Fanuc TP program (LS listing): mikado.ls

/PROG  MIKADO
/ATTR
OWNER		= MNEDITOR;
COMMENT		= "r3";
PROG_SIZE	= 270;
CREATE		= DATE 16-09-30  TIME 09:07:42;
MODIFIED	= DATE 16-10-04  TIME 11:47:18;
FILE_NAME	= ;
VERSION		= 0;
LINE_COUNT	= 6;
MEMORY_SIZE	= 650;
PROTECT		= READ_WRITE;
TCD:  STACK_SIZE	= 1000,
      TASK_PRIORITY	= 50,
      TIME_SLICE	= 0,
      BUSY_LAMP_OFF	= 0,
      ABORT_REQUEST	= 0,
      PAUSE_REQUEST	= 7;
DEFAULT_GROUP	= 1,*,*,*,*;
CONTROL_CODE	= 00000000 00000000;
/MN
	: ! reset blocker DOs before starting ;
	: DO[145] = OFF ;
	: DO[146] = OFF ;
	: RUN ROS_STATE ;
	: ! init user log screen takes some ;
	: WAIT    .30(sec) ;
	: RUN ROS_TRAJ ;
	: RUN ROS_IO ;
	: CALL ROS_MOVESM    ;
/POS
/END
